{attribute 'qualified_only'}
VAR_GLOBAL
	actual_velocity AT%I*: DINT;

	
	
	
END_VAR

(* stored: Version 1.1.0.1, ProductVersion 3.1.4024.4
   GVL Global_actual_velocity: Id {81e71619-22bd-4359-83b2-3e624603b444} *)
